// TIA Portal V17 export
// export: Created 2022-05-04T07:11:14.8990119Z, ExportSetting WithDefaults, DisplayName Totally Integrated Automation Portal, DisplayVersion V17 Update 3, DisplayName TIA Portal Openness, DisplayVersion V17 Update 3, DisplayName TIA Portal Teamcenter Gateway, DisplayVersion V17 Update 3, DisplayName TIA Portal Version Control Interface, DisplayVersion V17, DisplayName SINAMICS Startdrive Advanced, DisplayVersion V17 Update2, DisplayName SINAMICS Startdrive G130, G150, S120, S150, SINAMICS MV, S210, DisplayVersion V17 Update2, DisplayName SINAMICS Startdrive G110M, G120, G120C, G120D, G120P, G115D, DisplayVersion V17 Update2, DisplayName STEP 7 Professional, DisplayVersion V17 Update 3, DisplayName STEP 7 CFC, DisplayVersion V17 Update 1, DisplayName STEP 7 Safety, DisplayVersion V17, DisplayName WinCC UA Professional, DisplayVersion V17 Update 3, DisplayName WinCC Unified Calendar, DisplayVersion V17, DisplayName WinCC Unified Performance Insight, DisplayVersion V17
DATA_BLOCK "IDB_RK512_on_TCP"   // DB5
AUTHOR : G.DEJEAN
FAMILY : Comm
NAME : RK_TCPIP
VERSION : 0.1
// stored: AutoNumber true, DBAccessibleFromOPCUA true, DBAccessibleFromWebserver true, InstanceOfName RK512_on_TCP, InstanceOfType FB
"RK512_on_TCP"
   // VAR_INPUT
   //    HW_ID : HW_ANY;
   //    Local_Port : UInt;
   // END_VAR
   // VAR_OUTPUT
   //    Status_Conn_TCP : Word;
   //    Status_RK512 : Word;
   // END_VAR
   // VAR_IN_OUT
   //    Init : Bool;
   // END_VAR
   // VAR
   //    Attente_Data { ExternalAccessible := 'False'; ExternalVisible := 'False'; ExternalWritable := 'False'} : Bool;
   //    Attente_STX { ExternalAccessible := 'False'; ExternalVisible := 'False'; ExternalWritable := 'False'} : Bool;
   //    "Step" { ExternalAccessible := 'False'; ExternalVisible := 'False'; ExternalWritable := 'False'} : Int;
   //    LEN_RECEPTION_TCP : UDInt;
   //    LEN_EMISSION_TCP : UDInt;
   //    Long_Transfert { ExternalAccessible := 'False'; ExternalVisible := 'False'; ExternalWritable := 'False'} : Word;
   //    Long_Transfert_suite { ExternalAccessible := 'False'; ExternalVisible := 'False'; ExternalWritable := 'False'} : Word;
   //    REQ_Emission : Bool;
   //    Time_Out_Recep_Data : Bool;
   //    Fin_attente_Emis_STX : Bool;
   //    Flag_SEND : Bool;
   //    Flag_SEND_SUITE : Bool;
   //    Flag_FETCH : Bool;
   //    Flag_FETCH_SUITE : Bool;
   //    Flag_FETCH_SUITE_END : Bool;
   //    Flag_SEND_END : Bool;
   //    Flag_FETCH_END : Bool;
   //    Save_DWNR_suite : Byte;
   //    Save_DBNR_suite : Byte;
   //    CONNECT_TCP { S7_SetPoint := 'True'} : TCON_IP_v4;
   //    RECEPTION_TCP : Array[1..256] of Byte;
   //    EMISSION_TCP : Array[1..256] of Byte;
   //    Buffer_datas { ExternalAccessible := 'False'; ExternalVisible := 'False'; ExternalWritable := 'False'} : Array[1..256] of Byte;
   //    TRCV_C_Instance { S7_SetPoint := 'True'} : TRCV_C;
   //    TSEND_C_Instance { S7_SetPoint := 'True'} : TSEND_C;
   //    IEC_Timer_0_Instance { S7_SetPoint := 'True'} : TON_TIME;
   //    IEC_Timer_1_Instance { S7_SetPoint := 'True'} : TON_TIME;
   // END_VAR
BEGIN
END_DATA_BLOCK
